{attribute 'hide_all_locals'}
FUNCTION_BLOCK DisableGroup IMPLEMENTS ITask
VAR_INPUT
END_VAR
VAR_OUTPUT
END_VAR
VAR
	groupDisable			: MC_GroupDisable;
	_caGroup			: ICollisionGroup;
	State: INT;
	_disableGroup : BOOL;
	_busy : BOOL;
	_error : BOOL;
	_done : BOOL;
	Logger : TcMessage_Ext;
END_VAR

CASE State OF
	0:
		IF _disableGroup THEN
			_done := FALSE;
			_error := FALSE;
			_busy := TRUE;
			groupDisable.Execute := TRUE;
			IF groupDisable.Busy THEN
				_disableGroup := FALSE;
				State := 10;
				logger.Send(TC_EVENTS.XtsCAGroupEvents.CAGroupDisabling,'');
			END_IF
		END_IF
	
	10:
		IF NOT groupDisable.Busy THEN
			IF groupDisable.Done THEN
				_done := TRUE;
				logger.Send(TC_EVENTS.XtsCAGroupEvents.CAGroupDisabled,'');
			ELSIF groupDisable.Error THEN
				_error := TRUE;
				logger.Send(TC_EVENTS.XtsCAGroupEvents.CAGroupDisableError,'');
			END_IF
			_busy := FALSE;
			groupDisable.Execute := false;
			State := 0;
		END_IF
END_CASE


groupDisable(AxesGroup := _caGroup.GroupRef);

METHOD Abort : BOOL
State := 0;
groupDisable.Execute := FALSE;
Abort := true;
END_METHOD

PROPERTY Busy : BOOL
GET
Busy := _busy;
END_GET
END_PROPERTY

PROPERTY Done : BOOL
GET
Done := _done;
END_GET
END_PROPERTY

PROPERTY Error : BOOL
GET
Error := _error;
END_GET
END_PROPERTY

METHOD Execute : BOOL
Execute := _disableGroup := TRUE;
END_METHOD

METHOD FB_init : BOOL
VAR_INPUT
	bInitRetains : BOOL; // if TRUE, the retain variables are initialized (warm start / cold start)
	bInCopyCode : BOOL;  // if TRUE, the instance afterwards gets moved into the copy code (online change)
	CAGroup : ICollisionGroup;
END_VAR
_caGroup := CAGroup;
END_METHOD

END_FUNCTION_BLOCK

(* stored: Version 1.1.0.1, ProductVersion 3.1.4024.11
   POU DisableGroup: Id {2efb7482-2869-4c33-92cf-4ab1172a1cdc}, SpecialFunc None
   Method Abort: Id {3e18b1e4-3090-4bb5-ab59-aa6e4e12c0ef}
   Property Busy: Id {4930380f-5f69-4c59-abf0-3f7e820d28fd}
   Get Get: Id {042e9807-eaa3-4683-b892-f125b1618e0d}
   Property Done: Id {87722ae3-44ad-4fea-8bac-fcd129197625}
   Get Get: Id {ea9bc1eb-4961-4b5b-9e40-37ce15fd5f5a}
   Property Error: Id {446c2ac5-d9c1-4731-9b12-a47c4879f72e}
   Get Get: Id {8191c214-596a-427a-89fd-c9835883ce5b}
   Method Execute: Id {75a1aef5-6794-4797-8c10-1d2b68a1a592}
   Method FB_init: Id {e1d9a681-04bb-4f12-84b2-adf3edd36752} *)
